{attribute 'linkalways'} 
{attribute 'no_explicit_call' := 'This FB is a CLASS and must be accessed using methods or properties'}
{attribute 'enable_dynamic_creation'}
FUNCTION_BLOCK _ETcVnRTrees EXTENDS EnumDatatypeBase
VAR
	localData : ETcVnRTrees;
	activeData : REFERENCE TO ETcVnRTrees;
	enumBaseDatatype : _UDINT(localData);
END_VAR

METHOD PRIVATE AddLocalEnumeration
VAR_INPUT
	Enumeration : T_MAXSTRING;
	Value : ETcVnRTrees;
END_VAR
AddEnumeration(Enumeration, Value);
END_METHOD

PROPERTY PUBLIC Address : PVOID
GET
Address := ADR(activeData);
END_GET
END_PROPERTY

METHOD PUBLIC ClearReference
VAR_INPUT
END_VAR
activeData REF= localData;
SetBaseDatatypeReference();
END_METHOD

METHOD PUBLIC Clone : I_Datatype
VAR
    pClone : POINTER TO _ETcVnRTrees;
END_VAR
pClone := __NEW(_ETcVnRTrees(InitialValue := Value));
Clone := pClone^;
END_METHOD

METHOD FB_init : BOOL
VAR_INPUT
	bInitRetains : BOOL; // if TRUE, the retain variables are initialized (warm start / cold start)
	bInCopyCode : BOOL;  // if TRUE, the instance afterwards gets moved into the copy code (online change)
	InitialValue : ETcVnRTrees;
END_VAR
localData := InitialValue;
AddBaseDatatype(enumBaseDatatype);
ClearReference();

AddLocalEnumeration('TCVN_RT_CLASSIFIER', ETcVnRTrees.TCVN_RT_CLASSIFIER);
AddLocalEnumeration('TCVN_RT_REGRESSOR', ETcVnRTrees.TCVN_RT_REGRESSOR);
END_METHOD

PROPERTY PUBLIC Identifier : T_MAXSTRING
GET
Identifier := 'ETcVnRTrees';
END_GET
END_PROPERTY

METHOD IsEnumeratorValueEqual : BOOL
VAR_INPUT
	Enumerator : I_KeyValueForwardEnumerator;
END_VAR
VAR
	storedValue : ETcVnRTrees;
END_VAR
IF NOT Enumerator.TryGet(storedValue) THEN
	RETURN;
END_IF

IsEnumeratorValueEqual := storedValue = activeData;
END_METHOD

METHOD PUBLIC MakeReferenceTo
VAR_INPUT
	ReferenceTarget : REFERENCE TO ETcVnRTrees;
END_VAR
activeData REF= ReferenceTarget;
SetBaseDatatypeReference();
END_METHOD

METHOD PROTECTED SetBaseDatatypeReference
VAR_INPUT
END_VAR
enumBaseDatatype.MakeReferenceTo(activeData);
END_METHOD

PROPERTY PUBLIC Size : UDINT
GET
Size := SIZEOF(activeData);
END_GET
END_PROPERTY

METHOD TryMakeReferenceTo : BOOL
VAR_INPUT
	Target : I_Datatype;
END_VAR
VAR
	targetAsEnum : I_EnumDatatype;
	pTargetData : POINTER TO ETcVnRTrees;
END_VAR
IF NOT Target.TryResolveAsEnumDatatype(targetAsEnum) THEN
	RETURN;
END_IF

IF targetAsEnum.Identifier <> Identifier THEN
	RETURN;
END_IF

pTargetData := Target.Address;
activeData REF= pTargetData^;
SetBaseDatatypeReference();
TryMakeReferenceTo := TRUE;
END_METHOD

PROPERTY PUBLIC Value : ETcVnRTrees
GET
Value := activeData;
END_GET
SET
activeData := Value;
END_SET
END_PROPERTY

END_FUNCTION_BLOCK

(* stored: Version 1.1.0.1, ProductVersion 3.1.4024.12
   POU _ETcVnRTrees: Id {cb2aca15-3dad-00c5-0a8e-a5b4882edeba}, SpecialFunc None
   Folder Constructor: Id {b7c7994b-5d13-0537-3d84-0f012c12034f}
   Folder Private: Id {184ea0aa-1460-0cea-3909-477cf985a8f4}
   Folder Protected: Id {6b6a72d3-2db2-0dc8-30ab-fa2376b8eb62}
   Method AddLocalEnumeration: Id {6aee14ff-1c3b-05b4-151e-49ccd90187f3}
   Property Address: Id {0b4ef5ef-4921-0dc3-35a8-d7d453b93459}
   Get Get: Id {32b56f94-dd9d-02cc-34b0-80696789e797}
   Method ClearReference: Id {5af24062-1ac1-0fb7-3ed5-1c59096f040a}
   Method Clone: Id {0ad21c1f-610a-07b9-3a23-f06f02d7ebd4}
   Method FB_init: Id {f35bc8c3-df1e-0be7-13dc-13036a8b956d}
   Property Identifier: Id {cad4181f-3117-0050-18fb-e016d7c09982}
   Get Get: Id {aa0c81ff-facd-03ab-1527-7a6235743d9c}
   Method IsEnumeratorValueEqual: Id {6c00c8c4-fd77-07db-38d0-a20d1e4466dc}
   Method MakeReferenceTo: Id {00dad150-495d-025d-033b-c4edd7d96194}
   Method SetBaseDatatypeReference: Id {194c4d82-0bbe-0257-3977-ce713e844faa}
   Property Size: Id {e41bc5f0-d9f1-0705-39b4-16950a8a2797}
   Get Get: Id {eac309a5-cf8a-0ef3-2d45-512d479f5c09}
   Method TryMakeReferenceTo: Id {823231f6-b72a-0b32-03cc-8e7fe5819fdd}
   Property Value: Id {2d7654ff-92bf-0318-0376-65ea2b3a2391}
   Get Get: Id {32a4429b-506d-013d-0169-0ba67ca9b5dc}
   Set Set: Id {0588510d-0b42-01ed-06b6-364343704a5d} *)
